// TIA Portal V19 export
TYPE "LEXCHANGETRAY_typeAxisSimpleControlInterface_2"
// stored: Access Published
   STRUCT
      commandConfiguration { S7_SetPoint := 'True'} : "LEXCHANGETRAY_typeAxisSimpleControlCommandConfiguration2";
      commands { S7_SetPoint := 'True'} : "LEXCHANGETRAY_typeAxisSimpleControlCommands_2";
      monitoring { S7_SetPoint := 'True'} : "LEXCHANGETRAY_typeAxisSimpleControlProcessValues_2";
      configuration { S7_SetPoint := 'True'} : "LBC_typeAxisSimpleControlConfiguration";
   END_STRUCT;
END_TYPE
